// TIA Portal V17 export
// export: Created 2023-12-22T15:05:26.9882242Z, ExportSetting WithDefaults, DisplayName Totally Integrated Automation Portal, DisplayVersion V17, DisplayName TIA Portal Openness, DisplayVersion V17, DisplayName TIA Portal Version Control Interface, DisplayVersion V17, DisplayName STEP 7 Professional, DisplayVersion V17, DisplayName STEP 7 Safety, DisplayVersion V17, DisplayName WinCC Advanced, DisplayVersion V17
FUNCTION_BLOCK "DI_ex"   // FB101, LAD
{ S7_Optimized_Access := 'FALSE' }
VERSION : 0.1
// stored: AutoNumber false, IsIECCheckEnabled false, SetENOAutomatically false, UDAEnableTagReadback false
   VAR_INPUT
      I : Bool;   // Входной сигнал ПЛК
   END_VAR
   VAR_OUTPUT
      Signal : Bool;   // Результат обработки
   END_VAR
   VAR DB_SPECIFIC
      CMD : "CMD";   // Основные команды / Блок команд
      Use : Struct
         Inverse { S7_SetPoint := 'True'} : Bool;   // Инверсия входного сигнала
         Indirect { S7_SetPoint := 'True'} : Bool := true;   // Использование косвенной адресации
      END_STRUCT;
      ADDR_Byte { S7_SetPoint := 'True'} : Int;   // Адрес входа на контроллере (Байт)
      ADDR_Bit { S7_SetPoint := 'True'} : Int := 9;   // Адрес входа на контроллере (Бит)
   END_VAR
   VAR
      Filter_On { S7_SetPoint := 'True'} : "Time_S_b";   // Фильтр наличия сигнала
      Filter_Off { S7_SetPoint := 'True'} : "Time_S_b";   // Фильтр отсутствия сигнала
   END_VAR
   VAR_TEMP
      Data : Bool;
   END_VAR
   VAR_TEMP   // added for the SCL form of the ladder/FBD networks
      _w1 : Bool;
      _w2 : Bool;
   END_VAR
BEGIN

REGION Network 1: Устройство в ручном режиме
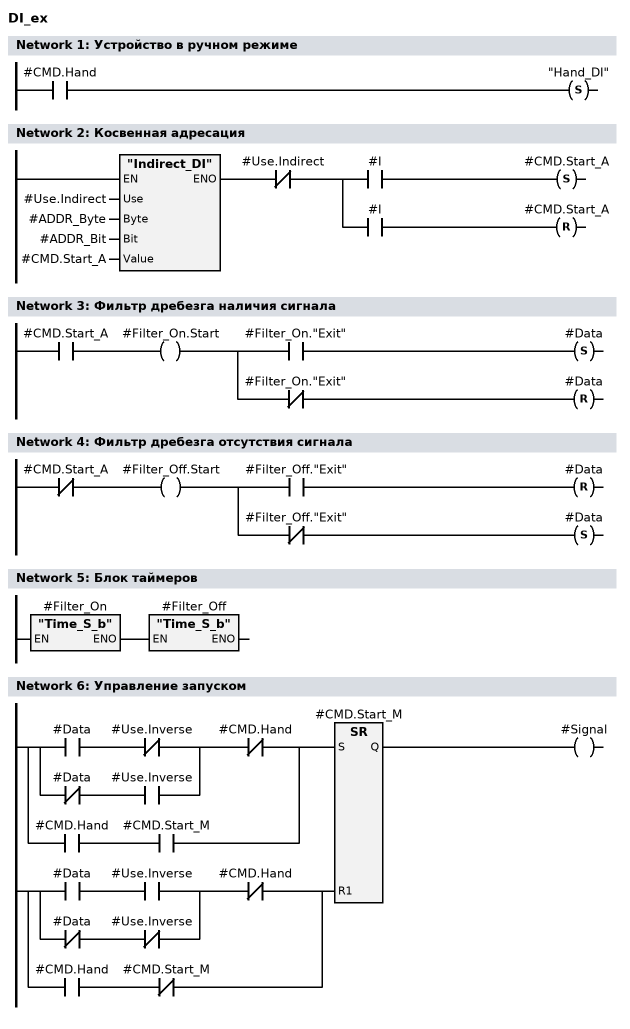
   RUNG wire#powerrail
      Contact( #CMD.Hand )
      S_Coil( "Hand_DI" )
   END_RUNG
   // the same network as SCL:
   IF #CMD.Hand THEN "Hand_DI" := TRUE; END_IF;
END_REGION

REGION Network 2: Косвенная адресация
   RUNG wire#powerrail
      "Indirect_DI"(Use := #Use.Indirect, "Byte" := #ADDR_Byte, Bit := #ADDR_Bit, Value := #CMD.Start_A)
      I_Contact( #Use.Indirect )
      wire#w1
      Contact( #I )
      S_Coil( #CMD.Start_A )
   END_RUNG
   RUNG wire#w1
      Contact( #I )
      R_Coil( #CMD.Start_A )
   END_RUNG
   // the same network as SCL:
   "Indirect_DI"(Use := #Use.Indirect,
                 "Byte" := #ADDR_Byte,
                 Bit := #ADDR_Bit,
                 Value := #CMD.Start_A,
                 ENO => #_w1);
   #_w2 := #_w1 AND NOT #Use.Indirect;
   IF #_w2 AND #I THEN
       #CMD.Start_A := TRUE;
       #CMD.Start_A := FALSE;
   END_IF;
END_REGION

REGION Network 3: Фильтр дребезга наличия сигнала
   RUNG wire#powerrail
      Contact( #CMD.Start_A )
      Coil( #Filter_On.Start )
      wire#w1
      Contact( #Filter_On."Exit" )
      S_Coil( #Data )
   END_RUNG
   RUNG wire#w1
      I_Contact( #Filter_On."Exit" )
      R_Coil( #Data )
   END_RUNG
   // the same network as SCL:
   #Filter_On.Start := #CMD.Start_A;
   IF #CMD.Start_A AND #Filter_On."Exit" THEN #Data := TRUE; END_IF;
   IF #CMD.Start_A AND NOT #Filter_On."Exit" THEN #Data := FALSE; END_IF;
END_REGION

REGION Network 4: Фильтр дребезга отсутствия сигнала
   RUNG wire#powerrail
      I_Contact( #CMD.Start_A )
      Coil( #Filter_Off.Start )
      wire#w1
      Contact( #Filter_Off."Exit" )
      R_Coil( #Data )
   END_RUNG
   RUNG wire#w1
      I_Contact( #Filter_Off."Exit" )
      S_Coil( #Data )
   END_RUNG
   // the same network as SCL:
   #Filter_Off.Start := NOT #CMD.Start_A;
   IF NOT #CMD.Start_A AND #Filter_Off."Exit" THEN #Data := FALSE; END_IF;
   IF NOT #CMD.Start_A AND NOT #Filter_Off."Exit" THEN #Data := TRUE; END_IF;
END_REGION

REGION Network 5: Блок таймеров
   RUNG wire#powerrail
      #Filter_On()
      #Filter_Off()
   END_RUNG
   // the same network as SCL:
   #Filter_On(ENO => #_w1);   // "Time_S_b"
   IF #_w1 THEN
       #Filter_Off();   // "Time_S_b"
   END_IF;
END_REGION

REGION Network 6: Управление запуском
   RUNG wire#powerrail
      Contact( #Data )
      I_Contact( #Use.Inverse )
      wire#w1
      I_Contact( #CMD.Hand )
      wire#w2
      S_SR(operand := #CMD.Start_M, r1 := wire#w4)
      Coil( #Signal )
   END_RUNG
   RUNG wire#powerrail
      I_Contact( #Data )
      Contact( #Use.Inverse )
   END_RUNG wire#w1
   RUNG wire#powerrail
      Contact( #CMD.Hand )
      Contact( #CMD.Start_M )
   END_RUNG wire#w2
   RUNG wire#powerrail
      Contact( #Data )
      Contact( #Use.Inverse )
      wire#w3
      I_Contact( #CMD.Hand )
   END_RUNG wire#w4
   RUNG wire#powerrail
      I_Contact( #Data )
      I_Contact( #Use.Inverse )
   END_RUNG wire#w3
   RUNG wire#powerrail
      Contact( #CMD.Hand )
      I_Contact( #CMD.Start_M )
   END_RUNG wire#w4
   // the same network as SCL:
   #_w1 := (((#Data AND #Use.Inverse) OR (NOT #Data AND NOT #Use.Inverse)) AND NOT #CMD.Hand) OR (#CMD.Hand AND NOT #CMD.Start_M);
   IF (((#Data AND NOT #Use.Inverse) OR (NOT #Data AND #Use.Inverse)) AND NOT #CMD.Hand) OR (#CMD.Hand AND #CMD.Start_M) THEN
       #CMD.Start_M := TRUE;   // SR flip-flop
   END_IF;
   IF #_w1 THEN #CMD.Start_M := FALSE; END_IF;
   #Signal := #CMD.Start_M;
END_REGION
END_FUNCTION_BLOCK
